(* CoDeSys 2.3.9.31 project: 2floor.5.pr6 *)
(* Author: Yurko Shybaigolova *)
(* Libraries: TcAdsBC.lb6 5.7.02 12:03:02, PlcHelperBC.lb6 7.5.01 12:03:00, TcKL6301.lb6*6.9.12 16:26:00, STANDARD.LB6 5.6.98 12:03:02 *)

(* Global variable list: main *)
VAR_GLOBAL
(*ADS*)
	ads_adr1: STRING:='10.0.5.61.1.1';
	ads_adr2: STRING:='10.0.5.62.1.1';
	ads_adr3: STRING:='10.0.5.63.1.1';

	write_ads: ADSWRITE;
	close_ads:ADSCLOSE;
	read_ads1: ADSREADEX;
	read_ads3: ADSREADEX;

	data1floor: ARRAY[0..4] OF BYTE;
	data1floor_prev: ARRAY[0..4] OF BYTE;


	m_fancoil_kabinet_low 	AT%MX0.0: BOOL;
	m_fancoil_kabinet_med 	AT%MX0.1: BOOL;
	m_fancoil_kabinet_high 	AT%MX0.2: BOOL;
	m_collector				AT%MB1:BYTE;
	m_klapan_kabinet		AT%MW2: WORD;

	m_fancoil_kino_low 		AT%MX0.3: BOOL;
	m_fancoil_kino_med 	AT%MX0.4: BOOL;
	m_fancoil_kino_high		AT%MX0.5: BOOL;

	kabinet_shtory			AT%MX7.0:BOOL;
	kabinet_tul				AT%MX7.1:BOOL;
	kino_shtory				AT%MX7.2:BOOL;
	kino_tul					AT%MX7.3:BOOL;


	m_klapan_kino			AT%MW4: WORD;


	skhody3				AT%MX6.0:BOOL;
	skhody1				AT%MX10.0:BOOL;






END_VAR

(* Global variable list: physical *)
VAR_GLOBAL
	din1_1	AT %IX52.0:	BOOL;
	din1_2	AT %IX52.1:	BOOL;
	din1_3	AT %IX52.2:	BOOL;
	din1_4	AT %IX52.3:	BOOL;
	din1_5	AT %IX52.4:	BOOL;
	din1_6	AT %IX52.5:	BOOL;
	din1_7	AT %IX52.6:	BOOL;
	din1_8	AT %IX52.7:	BOOL;
	din2_1	AT %IX53.0:	BOOL;
	din2_2	AT %IX53.1:	BOOL;
	din2_3	AT %IX53.2:	BOOL;
	din2_4	AT %IX53.3:	BOOL;
	din2_5	AT %IX53.4:	BOOL;
	din2_6	AT %IX53.5:	BOOL;
	din2_7	AT %IX53.6:	BOOL;
	din2_8	AT %IX53.7:	BOOL;
(*din3_1*)sw_kino_balkon	AT %IX54.0:	BOOL;
(*din3_2*)sw_tambur2		AT %IX54.1:	BOOL;
(*din3_3*)sw_kino1			AT %IX54.2:	BOOL;
(*din3_4*)sw_korydor		AT %IX54.3:	BOOL;
(*din3_5*)sw_kino2			AT %IX54.4:	BOOL;
(*din3_6*)sw_studio1			AT %IX54.5:	BOOL;
(*din3_7*)sw_tambur1		AT %IX54.6:	BOOL;
(*din3_8*)sw_studio2			AT %IX54.7:	BOOL;
(*din4_1*)sw_kabinet1		AT %IX55.0:	BOOL;
	din4_2	AT %IX55.1:	BOOL;
(*din4_3*)sw_kabinet2	AT %IX55.2:	BOOL;
(*din4_4*)sw_kabinet2_1	AT %IX55.3:	BOOL;
(*din4_5*)sw_kabinet_balkon	AT %IX55.4:	BOOL;
(*din4_6*)sw_kabinet2_2	AT %IX55.5:	BOOL;
(*din4_7*)sw_tambur3		AT %IX55.6:	BOOL;
	din4_8	AT %IX55.7:	BOOL;

(*dout1_1*)balkon_peryla				AT %QX52.0:	BOOL;
(*dout1_2*)kino_l					AT %QX52.1:	BOOL;
(*dout1_3*)balkon_bra				AT %QX52.2:	BOOL;
(*dout1_4*)kabinet_balkon_l			AT %QX52.3:	BOOL;
(*dout1_5*)balkon					AT %QX52.4:	BOOL;
(*dout1_6*)korydor1					AT %QX52.5:	BOOL;
(*dout1_7*)kino_bra					AT %QX52.6:	BOOL;
(*dout1_8*)korydor2					AT %QX52.7:	BOOL;
(*dout2_1*)studio_pidsvitka 			AT %QX53.0:	BOOL;
(*dout2_2*)skhody2_3				AT %QX53.1:	BOOL;
(*dout2_3*)studio_l					AT %QX53.2:	BOOL;
(*dout2_4*)kabinet_pidsvitka_kolo	AT %QX53.3:	BOOL;
(*dout2_5*)kabinet_svitlo				AT %QX53.4:	BOOL;
(*dout2_6*)kabinet_kobra 			AT %QX53.5:	BOOL;
(*dout2_7*)tambur_l					AT %QX53.6:	BOOL;
	stend	AT %QX53.7:	BOOL;
(*dout3_1*)collector_kabinet1		AT %QX54.0:	BOOL;
(*dout3_2*)fancoil_kabinet_low		AT %QX54.1:	BOOL;
(*dout3_3*)collector_kabinet2		AT %QX54.2:	BOOL;
(*dout3_4*)fancoil_kabinet_med		AT %QX54.3:	BOOL;
(*dout3_5*)collector_studio1			AT %QX54.4:	BOOL;
	fancoil_kabinet_high				AT %QX54.5:	BOOL;
(*dout3_7*)collector_studio2			AT %QX54.6:	BOOL;
(*dout3_8*)fancoil_kino_low			AT %QX54.7:	BOOL;
(*dout4_1*)fancoil_kino_med		AT %QX55.0:	BOOL;
	dout4_2	AT %QX55.1:	BOOL;
	fancoil_kino_high				AT %QX55.2:	BOOL;
	skhody_peryla	AT %QX55.3:	BOOL;
	dout4_5	AT %QX55.4:	BOOL;
	dout4_6	AT %QX55.5:	BOOL;
	dout4_7	AT %QX55.6:	BOOL;
	dout4_8	AT %QX55.7:	BOOL;
	kino_tul_open			AT %QX56.0:	BOOL;
	kabinet_tul_close 		AT %QX56.1:	BOOL;
	kino_tul_close 			AT %QX56.2:	BOOL;
	kabinet_tul_open		AT %QX56.3:	BOOL;
	kino_shtory_open		AT %QX56.4:	BOOL;
	kabinet_shtory_open	AT %QX56.5:	BOOL;
	kino_shtory_close		AT %QX56.6:	BOOL;
	kabinet_shtory_close	AT %QX56.7:	BOOL;


	klapan_kino 	AT %QB2:	INT;
	klapan_kabinet	AT %QB6:	INT; (*0-opened, 16#7fff - closed*)

	temp_kabinet	AT %IB18:	INT;
	temp_studio		 AT %IB26:	INT;


	Term_12_KL3228_4_1_State	AT %IB16:	USINT;

	Term_12_KL3228_4_1_Ctrl	AT %QB16:	USINT;
	Term_12_KL3228_4_1_Data_Out	AT %QB18:	INT;
	Term_12_KL3228_4_2_State	AT %IB20:	USINT;
	Term_12_KL3228_4_2_Data_In	AT %IB22:	INT;
	Term_12_KL3228_4_2_Ctrl	AT %QB20:	USINT;
	Term_12_KL3228_4_2_Data_Out	AT %QB22:	INT;
	Term_12_KL3228_4_3_State	AT %IB24:	USINT;

	Term_12_KL3228_4_3_Ctrl	AT %QB24:	USINT;
	Term_12_KL3228_4_3_Data_Out	AT %QB26:	INT;
	Term_12_KL3228_4_4_State	AT %IB28:	USINT;
	Term_12_KL3228_4_4_Data_In	AT %IB30:	INT;
	Term_12_KL3228_4_4_Ctrl	AT %QB28:	USINT;
	Term_12_KL3228_4_4_Data_Out	AT %QB30:	INT;
	Term_13_KL3228_4_1_State	AT %IB32:	USINT;
	Term_13_KL3228_4_1_Data_In	AT %IB34:	INT;
	Term_13_KL3228_4_1_Ctrl	AT %QB32:	USINT;
	Term_13_KL3228_4_1_Data_Out	AT %QB34:	INT;
	Term_13_KL3228_4_2_State	AT %IB36:	USINT;
	Term_13_KL3228_4_2_Data_In	AT %IB38:	INT;
	Term_13_KL3228_4_2_Ctrl	AT %QB36:	USINT;
	Term_13_KL3228_4_2_Data_Out	AT %QB38:	INT;
	Term_13_KL3228_4_3_State	AT %IB40:	USINT;
	Term_13_KL3228_4_3_Data_In	AT %IB42:	INT;
	Term_13_KL3228_4_3_Ctrl	AT %QB40:	USINT;
	Term_13_KL3228_4_3_Data_Out	AT %QB42:	INT;
	Term_13_KL3228_4_4_State	AT %IB44:	USINT;
	Term_13_KL3228_4_4_Data_In	AT %IB46:	INT;
	Term_13_KL3228_4_4_Ctrl	AT %QB44:	USINT;
	Term_13_KL3228_4_4_Data_Out	AT %QB46:	INT;
	Term_14_KL2761_State	AT %IB48:	USINT;
	Term_14_KL2761_Data_In	AT %IB50:	INT;
	Term_14_KL2761_Ctrl	AT %QB48:	USINT;
	Term_14_KL2761_Data_Out	AT %QB50:	INT;



END_VAR

(* POU MAIN, ST *)
PROGRAM MAIN
VAR

END_VAR
light;
heat;
shtory_kino;
shtory_kabinet;
ADS_write;
END_PROGRAM

(* POU light, ST *)
PROGRAM light
VAR
	kino_balkon, kino1, kino2, studio1,studio2, kabinet1, kabinet2, kabinet_balkon, korydor, tambur1, tambur2, tambur3: SWITCH;
	switch_delay: TIME;
	off_delay: TIME;

	SKHODY_R: R_TRIG;
	SKHODY_F: F_TRIG;
END_VAR
switch_delay:=t#500ms; (*затримка довгого натискання*)
off_delay:=t#3m; (*затримка для відкладеного вимкнення*)

kino_balkon(MODE:='short&long', IN:=sw_kino_balkon,SWITCH_DELAY:=switch_delay, Q_SHORT=>balkon, Q_LONG=>balkon_bra);
balkon_peryla:=kino_balkon.Q_LONG;

kino1(MODE:='short&long',IN:=sw_kino1, SWITCH_DELAY:=switch_delay, Q_SHORT=>kino_l);
kino2(MODE:='short&long', IN:=sw_kino2, SWITCH_DELAY:=switch_delay, Q_SHORT=>kino_bra);
studio1(MODE:='short&long', IN:=sw_studio1, SWITCH_DELAY:=switch_delay, Q_SHORT=>studio_l);
studio2(MODE:='short&long', IN:=sw_studio2, SWITCH_DELAY:=switch_delay, Q_SHORT=>studio_pidsvitka);

korydor(MODE:='short&long', IN:=sw_korydor, SWITCH_DELAY:=switch_delay);
korydor1:=korydor.Q_SHORT;
korydor2:=korydor.Q_SHORT;

kabinet1(MODE:='short&long', IN:=sw_kabinet1 XOR sw_kabinet2_1, SWITCH_DELAY:=switch_delay, Q_SHORT=>kabinet_svitlo);

kabinet2(MODE:='short&long', IN:=sw_kabinet2 XOR sw_kabinet2_2, SWITCH_DELAY:=switch_delay);
kabinet_kobra:=kabinet2.Q_SHORT;
kabinet_pidsvitka_kolo:=kabinet2.Q_SHORT;

kabinet_balkon(MODE:='short&long', IN:=sw_kabinet_balkon, SWITCH_DELAY:=switch_delay, Q_SHORT=>kabinet_balkon_l);

tambur3(MODE:='short&long', IN:=sw_tambur3, SWITCH_DELAY:=switch_delay, Q_SHORT=>stend);



(*відстежую натискання вимикачів на обох поверхах і перемикаю лампочку по кожному натисненні*)
SKHODY_R(CLK:=skhody1 XOR skhody3 XOR sw_tambur1);

IF SKHODY_R.Q OR SKHODY_F.Q THEN skhody2_3:= NOT skhody2_3; END_IF
skhody_peryla:=skhody2_3;
data1floor[0].0:=sw_tambur1 ;
END_PROGRAM

(* POU Vymykachi/SWITCH, ST *)
FUNCTION_BLOCK SWITCH
VAR_INPUT
	IN:BOOL;
	SWITCH_DELAY:TIME; (*різниця між коротким і довгим натисненням*)
	SHORT_OFF_DELAY, LONG_OFF_DELAY: TIME; (*час затримки вимкнення по короткому та довгому натисненню*)
	MODE:STRING; (*delayed, light, light&vent, short&long, delayed_short&long, *)
	NUMBER_OF_OUTS:INT;
END_VAR
VAR_OUTPUT
	Q_SHORT:BOOL:=FALSE;
	Q_SHORT_D: BOOL;(*вихід для вимкнення із затримкою, вмикається разом із виходом короткого натискання*)
	Q_LONG:BOOL:=FALSE;
	Q_LONG_D:BOOL; (*вихід для вимкнення із затримкою, вмикається разом із виходом довгого натискання*)
END_VAR
VAR
	STAN:BOOL:=FALSE;
	Q_S_fall:F_TRIG; (*ловить задній фронт вихода короткого натискання*)
	Q_L_fall:F_TRIG;(*ловить задній фронт вихода довгого натискання*)
	chas: TIME; (*час доки кнопка натиснена*)

	long: BOOL; (*стає тру, якщо було довге натиснення*)
	short: BOOL; (*стає тру, якщо було коротке натиснення*)
	timer, short_off_delay_timer, long_off_delay_timer: TON; (*таймери: час натискання, час переключення відкладеного виходу по довгому та короткому натисканнях*)
	up: BOOL; (*кнопка натиснена*)

	delay_l, delay_s:BOOL; (*запускати таймери відкладеного вимкнення*)

	turn_off_long: BOOL;
	start_l, start_s:BOOL;
END_VAR
short:=0;
long:=0;
timer(IN:=IN AND STAN, PT:=t#10s);
IF IN AND STAN THEN
	chas:=timer.ET;
	up:=1;
ELSE
up:=0;
END_IF;

IF NOT IN AND NOT STAN THEN
chas:=t#0ms;
END_IF;

IF STAN AND NOT IN THEN
	IF chas <SWITCH_DELAY THEN
		short:=1;
		Q_SHORT:= NOT Q_SHORT;
	END_IF;
	IF chas>=SWITCH_DELAY THEN
		Q_LONG:= NOT Q_LONG;
		long:=1;
	END_IF;
END_IF;

(*затримка вимикання*)
Q_L_fall(CLK:=Q_LONG);
Q_S_fall(CLK:=Q_SHORT);

IF Q_L_FALL.Q THEN
		start_l:=TRUE;
END_IF

IF Q_S_FALL.Q THEN
	start_s:=TRUE;
END_IF

IF MODE='light&vent' THEN
	IF start_s THEN start_l:=start_s; END_IF
END_IF

IF LONG_OFF_DELAY <> t#0ms THEN (*виконувати лише якщо в блок переданий параметр затримки на вимкнення*)

	IF Q_LONG THEN
		Q_LONG_D:=Q_LONG;
	END_IF

	long_off_delay_timer(IN:=start_l, PT:=LONG_OFF_DELAY);

	IF long_off_delay_timer.Q THEN
		Q_LONG_D:=FALSE;
		start_l:=FALSE;
	END_IF

ELSE
	Q_LONG_D:=Q_LONG;
END_IF

IF SHORT_OFF_DELAY <> t#0ms THEN (*виконувати лише якщо в блок переданий параметр затримки на вимкнення*)

	IF Q_SHORT THEN
		Q_SHORT_D:=Q_SHORT;
	END_IF

	short_off_delay_timer(IN:=start_s, PT:=SHORT_OFF_DELAY);

	IF short_off_delay_timer.Q THEN
		Q_SHORT_D:=FALSE;
		start_s:=FALSE;
	END_IF


ELSE
	Q_SHORT_D:=Q_SHORT;
END_IF

IF MODE='delayed' THEN
	Q_LONG:=Q_LONG_D;
	Q_SHORT:=Q_SHORT_D;
END_IF
(*працють лише короткі замикання*)
IF MODE='light' THEN
	Q_SHORT_D:=FALSE;
	Q_LONG:=Q_SHORT;
	Q_LONG_D:=FALSE;
END_IF
(*затримки не працюють*)
IF MODE='short&long' THEN
	Q_SHORT_D:=FALSE;
	Q_LONG_D:=FALSE;
END_IF
(*при вимкненні всього світла вимикати вентилятор і затримкою*)
IF MODE='light&vent' THEN
	IF NOT Q_SHORT AND Q_LONG THEN
		Q_LONG:=Q_LONG_D;
	END_IF
END_IF

STAN := IN;
END_FUNCTION_BLOCK

(* POU heat, ST *)
PROGRAM heat
VAR
	fancoil_kino: WORD;
	fancoil_kabinet:  WORD;

END_VAR
	fancoil_kino_low:=m_fancoil_kino_low;
	fancoil_kino_med:=m_fancoil_kino_med;
	fancoil_kino_high:=m_fancoil_kino_high;
	klapan_kino:=m_klapan_kino;

	fancoil_kabinet_low:=m_fancoil_kabinet_low;
	fancoil_kabinet_med:=m_fancoil_kabinet_med;
	fancoil_kabinet_high:=m_fancoil_kabinet_high;
	klapan_kabinet:=m_klapan_kabinet;

collector_kabinet1:=m_collector.0;
collector_kabinet2:=m_collector.1;
collector_studio1:=m_collector.2;
collector_studio2:=m_collector.3;
END_PROGRAM

(* POU shtory_kino, ST *)
PROGRAM shtory_kino
VAR
	inc1, inc: UINT;
	impulse: BOOL;
	shtory_status: BOOL;(*1 - closed, 0 - opened*)
	impulse1: BOOL;
	tul_status: BOOL;(*1 - closed, 0 - opened*)
	lift_move_dir, lift_moves: BOOL;
	rising1: BOOL;
	falling1: BOOL;
	rising2: BOOL;
	falling2: BOOL;
	inc2: UINT;
	panel_shtory_move, panel_tul_move :BOOL;

	(*таймери для формування керуючих імпульсів*)
	timer_shtory_move, timer_shtory_stop,timer_tul_move, timer_tul_stop, move_lift_up, move_lift_down: TP;

	shtory_counter, tul_counter, lift_counter: UINT;
	counter:CTU;

	shtory_move: BOOL;
	shtory_stop: BOOL;
	tul_move: BOOL;
	eib_tul_move: BOOL;
	eib_shtory_move: BOOL;
	R_SHTORY:R_TRIG;
	F_SHTORY:F_TRIG;
	R_TUL:R_TRIG;
	F_TUL:F_TRIG;

END_VAR
(*детекція відсутності фронтів*)
IF light.kino1.Q_LONG = impulse THEN
	rising1:=0;
	falling1:=0;
END_IF;

IF light.kino2.Q_LONG = impulse1 THEN
	rising2:=0;
	falling2:=0;
END_IF;

(*ловим передній фронт довгого натискання першої клавіші*)
IF light.kino1.Q_LONG AND NOT impulse  THEN
	rising1:=1;
	falling1:=0;
END_IF;

(*задній фронт*)
IF NOT light.kino1.Q_LONG AND  impulse THEN
	falling1:=1;
	rising1:=0;
END_IF;

(*ловим передній фронт довгого натискання другої клавіші*)
IF light.kino2.Q_LONG AND NOT impulse1  THEN
	rising2:=1;
	falling2:=0;
END_IF;

(*ловим задній фронт довгого натискання другої клавіші*)
IF NOT light.kino2.Q_LONG AND  impulse1 THEN
	falling2:=1;
	rising2:=0;
END_IF;


(*команди шторам смарт баса на 3 поверсі*)
R_SHTORY(CLK:=kino_shtory, Q=>eib_shtory_move);
IF NOT R_SHTORY.Q THEN F_SHTORY(CLK:=kino_shtory, Q=>eib_shtory_move); END_IF

R_TUL(CLK:=kino_tul, Q=>eib_tul_move);
IF NOT R_TUL.Q THEN F_TUL(CLK:=kino_tul, Q=>eib_tul_move); END_IF


shtory_move:= rising1 OR falling1 OR eib_shtory_move;
tul_move:= rising2 OR falling2 OR eib_tul_move;

(*формування імпульсів для керування шторами, тюлями та ліфтом*)
timer_shtory_move(IN:=shtory_move, PT:=t#1500ms);
timer_shtory_stop(IN:=shtory_move , PT:=t#1500ms);
timer_tul_move(IN:=tul_move  , PT:=t#1500ms);
timer_tul_stop(IN:=tul_move , PT:=t#1500ms);

	(*вибір рухати чи зупинити  штори*)
	IF shtory_move THEN
		inc:=inc+1;
	END_IF;
	IF inc>2 THEN inc:=1; END_IF;

	(*вибір рухати чи зупинити  тюль*)
	IF tul_move THEN
		inc1:=inc1+1;
	END_IF;
	IF inc1>2 THEN inc1:=1; END_IF;

	CASE inc OF

	1:
		kino_shtory_open:=timer_shtory_move.Q; (*відкривати*)
		kino_shtory_close:= 0;
		shtory_status:=0;

	2:
		kino_shtory_close:=timer_shtory_move.Q;(*закривати*)
		kino_shtory_open:= 0;
		shtory_status:=1;

	END_CASE;

	CASE inc1 OF

	1:
		kino_tul_open:=timer_tul_move.Q; (*відкривати*)
		kino_tul_close:= 0;
		tul_status:=0;
	2:
		kino_tul_close:=timer_tul_move.Q;(*закривати*)
		kino_tul_open:= 0;
		tul_status:=1;

	END_CASE;


(*запам'ятовування стану довгого натискання для детекції фронтів*)

impulse:=light.kino1.Q_LONG;
impulse1:=light.kino2.Q_LONG;
END_PROGRAM

(* POU shtory_kabinet, ST *)
PROGRAM shtory_kabinet
VAR
	inc1, inc: UINT;
	impulse: BOOL;
	shtory_status: BOOL; (*1 - closed, 0 - opened*)
	impulse1: BOOL;
	tul_status: BOOL; (*1 - closed, 0 - opened*)
	lift_move_dir, lift_moves: BOOL;
	rising1: BOOL;
	falling1: BOOL;
	rising2: BOOL;
	falling2: BOOL;
	inc2: UINT;
	panel_shtory_move, panel_tul_move :BOOL;

	(*таймери для формування керуючих імпульсів*)
	timer_shtory_move, timer_shtory_stop,timer_tul_move, timer_tul_stop, move_lift_up, move_lift_down: TP;

	shtory_counter, tul_counter, lift_counter: UINT;
	counter:CTU;

	shtory_move: BOOL;
	shtory_stop: BOOL;
	tul_move: BOOL;
	eib_tul_move: BOOL;
	eib_shtory_move: BOOL;
	R_SHTORY:R_TRIG;
	F_SHTORY:F_TRIG;
	R_TUL:R_TRIG;
	F_TUL:F_TRIG;

END_VAR
(*детекція відсутності фронтів*)
IF light.kabinet1.Q_LONG = impulse THEN
	rising1:=0;
	falling1:=0;
END_IF;

IF light.kabinet2.Q_LONG = impulse1 THEN
	rising2:=0;
	falling2:=0;
END_IF;

(*ловим передній фронт довгого натискання першої клавіші*)
IF light.kabinet1.Q_LONG AND NOT impulse  THEN
	rising1:=1;
	falling1:=0;
END_IF;

(*задній фронт*)
IF NOT light.kabinet1.Q_LONG AND  impulse THEN
	falling1:=1;
	rising1:=0;
END_IF;

(*ловим передній фронт довгого натискання другої клавіші*)
IF light.kabinet2.Q_LONG AND NOT impulse1  THEN
	rising2:=1;
	falling2:=0;
END_IF;

(*ловим задній фронт довгого натискання другої клавіші*)
IF NOT light.kabinet2.Q_LONG AND  impulse1 THEN
	falling2:=1;
	rising2:=0;
END_IF;


(*команди шторам смарт баса на 3 поверсі*)
R_SHTORY(CLK:=kabinet_shtory, Q=>eib_shtory_move);
IF NOT R_SHTORY.Q THEN F_SHTORY(CLK:=kabinet_shtory, Q=>eib_shtory_move); END_IF

R_TUL(CLK:=kabinet_tul, Q=>eib_tul_move);
IF NOT R_TUL.Q THEN F_TUL(CLK:=kabinet_tul, Q=>eib_tul_move); END_IF

shtory_move:= rising1 OR falling1 OR eib_shtory_move;
tul_move:= rising2 OR falling2 OR eib_tul_move;

(*формування імпульсів для керування шторами, тюлями та ліфтом*)
timer_shtory_move(IN:=shtory_move, PT:=t#1000ms);
timer_shtory_stop(IN:=shtory_move , PT:=t#1000ms);
timer_tul_move(IN:=tul_move  , PT:=t#1000ms);
timer_tul_stop(IN:=tul_move , PT:=t#1000ms);

	(*вибір рухати чи зупинити  штори*)
	IF shtory_move THEN
		inc:=inc+1;
	END_IF;
	IF inc>2 THEN inc:=1; END_IF;

	(*вибір рухати чи зупинити  тюль*)
	IF tul_move THEN
		inc1:=inc1+1;
	END_IF;
	IF inc1>2 THEN inc1:=1; END_IF;

	CASE inc OF

	1:
		kabinet_shtory_open:=timer_shtory_move.Q; (*відкривати*)
		kabinet_shtory_close:= 0;
		shtory_status:=0;

	2:
		kabinet_shtory_close:=timer_shtory_move.Q;(*закривати*)
		kabinet_shtory_open:= 0;
		shtory_status:=1;

	END_CASE;

	CASE inc1 OF

	1:
		kabinet_tul_open:=timer_tul_move.Q; (*відкривати*)
		kabinet_tul_close:= 0;
		tul_status:=0;
	2:
		kabinet_tul_close:=timer_tul_move.Q;(*закривати*)
		kabinet_tul_open:= 0;
		tul_status:=1;

	END_CASE;


(*запам'ятовування стану довгого натискання для детекції фронтів*)

impulse:=light.kabinet1.Q_LONG;
impulse1:=light.kabinet2.Q_LONG;
END_PROGRAM

(* POU ADS_write, ST *)
PROGRAM ADS_write
VAR
	write_timeout: TIME;
	b_write1: BOOL;
	write_ads1: ADSWRITE;

	timer1:TP;
	errorcounter1, pack_c:CTU ;
	test_word: WORD;
	i1,j1: INT;
	data_changed: BOOL;
	try_again1: BOOL;
END_VAR
(*1floor*)
FOR i1:=0 TO (SIZEOF(data1floor))-1 DO
	IF data1floor[i1]<>data1floor_prev[i1] THEN
		b_write1:=TRUE;
		EXIT;
	ELSE
		b_write1:=FALSE;
	END_IF
END_FOR

IF try_again1 AND NOT timer1.Q THEN
	b_write1:=TRUE;
	try_again1:=FALSE;
END_IF


IF write_ads1.BUSY THEN b_write1:=FALSE; END_IF

	write_ads1(
		NETID:=ads_adr1,
		PORT:=800,
		IDXGRP:=16#4020,
		IDXOFFS:=2,
		WRITE:=b_write1,
		TMOUT:=t#5s,
		LEN:=SIZEOF(data1floor),
		SRCADDR:=ADR(data1floor));

IF write_ads1.ERR AND NOT timer1.Q THEN
	timer1.IN:=TRUE;
	try_again1:=TRUE;
END_IF
timer1(PT:=write_timeout);
timer1.IN:=FALSE;


FOR j1:=0 TO (SIZEOF(data1floor))-1 DO
	data1floor_prev[j1]:=data1floor[j1];
END_FOR
END_PROGRAM
